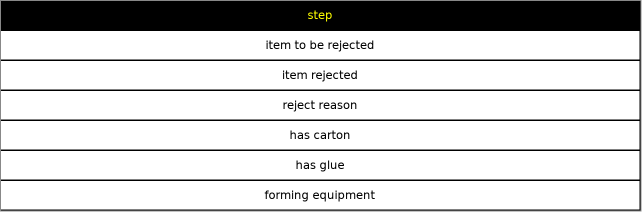
VISUALIZATION CARTON_FORMING_SHIFT_ELEMENT_DESCRIPTION  // 642x212
    Rectangle (0,0 640x30), "step"
    Rectangle (0,30 640x30), "item to be rejected"
    Rectangle (0,90 640x30), "reject reason"
    Rectangle (0,120 640x30), "has carton"
    Rectangle (0,180 640x30), "forming equipment"
    Rectangle (0,150 640x30), "has glue"
    Rectangle (0,60 640x30), "item rejected"
END_VISUALIZATION

(* stored: Version 1.1.0.1, ProductVersion 3.1.4024.3
   Visu CARTON_FORMING_SHIFT_ELEMENT_DESCRIPTION: Id {cbcd3cf9-a860-489b-9c27-c39238825c80} *)
